Yaskawa INFORM job: main_profile_long_22-06-23_planes_program.JBI

/JOB
//NAME main_profile_long_22-06-23_planes_program
//POS
///NPOS 4,0,4,0,0,0
///TOOL 0
///POSTYPE BASE
///RECTAN
///RCONF 0,0,0,0,0,0,0,0,0,0,0,0,0,0,0,0,0,0,0,0,0,0,0,0
///POSTYPE PULSE
///PULSE
//INST
///DATE 2023/06/22 16:21
///ATTR SC,RW,RJ
////FRAME BASE
///GROUP1 RB1,ST1
NOP
MOVJ P009 EX000 VJ=15.00
CALL JOB:SPYOF
MOVJ P009 VJ=15.00
CALL pos_z_0
MOVJ P009 VJ=15.00
CALL pos_z_1
MOVJ P009 VJ=15.00
CALL pos_z_2
MOVJ P009 VJ=15.00
END
